FUNCTION FC_Check_K : BOOL
VAR_INPUT
	I_sString : REFERENCE TO T_MaxString;
END_VAR
VAR
	stringPos	: INT;
END_VAR

stringPos := FIND(I_sString, 'K');
IF stringPos <> 0 THEN
	I_sString := MID(I_sString, LEN(I_sString), stringPos+1);
	FC_Check_K := TRUE;
ELSE
	FC_Check_K := FALSE;
END_IF

END_FUNCTION

(* stored: Version 1.1.0.1, ProductVersion 3.1.4024.15
   POU FC_Check_K: Id {8336332c-7d30-4622-afef-5111e653de63}, SpecialFunc None *)
